// TIA Portal project "FactoryIO_Template" (V16)
// Vorlageprojekt für das Buch mit Zielsystem S7-1200

(* hardware
DEVICE "S7-1200-Station_1"  S7-1200 Station
   slot 0: "Baugruppenträger_0"  Rack  V1.0
   slot 1: "PLC_1"  CPU 1211C DC/DC/DC  6ES7 211-1AE40-0XB0  V4.1
*)

// ===== PLC "PLC_1"  CPU 1211C DC/DC/DC =====

VAR_GLOBAL   // PLC tag table "Standard-Variablentabelle"
   "Sensor_1" AT %I0.3 : Bool;
   "Sensor_2" AT %I0.4 : Bool;
   "Sensor_3" AT %I0.5 : Bool;
   "Start_Button" AT %I0.0 : Bool;
   "Stop_Button" AT %I0.1 : Bool;
   "Reset_Button" AT %I0.2 : Bool;
   "Sensor_Input" AT %I0.6 : Bool;
   "Sensor_Output" AT %I0.7 : Bool;
   "Limit_0" AT %I1.0 : Bool;
   "Limit_90" AT %I1.1 : Bool;
   "Conveyor_1_(C1)" AT %Q0.0 : Bool;
   "Conveyor_2_(C2)" AT %Q0.1 : Bool;
   "Conveyor_3_(C3)" AT %Q0.2 : Bool;
   "Conveyor_4_(C4)" AT %Q0.3 : Bool;
   "Roll_(+)" AT %Q0.4 : Bool;
   "Roll_(-)" AT %Q0.5 : Bool;
   "Turn" AT %Q0.6 : Bool;
   "Start_Light" AT %Q0.7 : Bool;
   "Stop_Light" AT %Q1.0 : Bool;
   "Long_Counter" AT %QD40 : DInt;
   "Medium_Counter" AT %QD44 : DInt;
   "Short_Counter" AT %QD48 : DInt;
   "Long" AT %M1.0 : Bool;
   "Medium" AT %M1.1 : Bool;
   "Short" AT %M1.2 : Bool;
   "Emitter" AT %Q1.1 : Bool;
   "Read_Long_Counter" AT %MD0 : DInt;
   "Read_Medium_Counter" AT %MD4 : DInt;
   "Read_Short_Counter" AT %MD8 : DInt;
END_VAR

DATA_BLOCK "Phan_Loai_DB"   // DB1
{ S7_Optimized_Access := 'TRUE' }
VERSION : 0.1
// stored: InstanceOfName Phan_Loai
"Phan_Loai"
BEGIN
END_DATA_BLOCK

DATA_BLOCK "Control_DB"   // DB2
{ S7_Optimized_Access := 'TRUE' }
VERSION : 0.1
// stored: InstanceOfName Control
"Control"
BEGIN
END_DATA_BLOCK

// folder: System blocks/Program resources

DATA_BLOCK "Delay_500ms"   // DB3
{ S7_Optimized_Access := 'TRUE' }
AUTHOR : Simatic
FAMILY : IEC
NAME : IEC_TMR
VERSION : 1.0
// stored: InstanceOfName IEC_TIMER
"IEC_TIMER"
BEGIN
END_DATA_BLOCK

DATA_BLOCK "Counter_Long"   // DB4
{ S7_Optimized_Access := 'TRUE' }
AUTHOR : Simatic
FAMILY : IEC
NAME : CNTR
VERSION : 1.0
// stored: InstanceOfName IEC_COUNTER
"IEC_COUNTER"
BEGIN
END_DATA_BLOCK

DATA_BLOCK "Counter_Medium"   // DB5
{ S7_Optimized_Access := 'TRUE' }
AUTHOR : Simatic
FAMILY : IEC
NAME : CNTR
VERSION : 1.0
// stored: InstanceOfName IEC_COUNTER
"IEC_COUNTER"
BEGIN
END_DATA_BLOCK

DATA_BLOCK "Counter_Short"   // DB6
{ S7_Optimized_Access := 'TRUE' }
AUTHOR : Simatic
FAMILY : IEC
NAME : CNTR
VERSION : 1.0
// stored: InstanceOfName IEC_COUNTER
"IEC_COUNTER"
BEGIN
END_DATA_BLOCK

// folder: (top level)

FUNCTION_BLOCK "Phan_Loai"   // FB1, LAD
{ S7_Optimized_Access := 'TRUE' }
VERSION : 0.1
   VAR_INPUT
      SS1 : Bool;
      SS2 : Bool;
      SS3 : Bool;
   END_VAR
   VAR_OUTPUT
      Long : Bool;
      Medium : Bool;
      Short : Bool;
   END_VAR
   VAR
      Temp_Long : Bool;
      Temp_Medium : Bool;
      Temp_Short : Bool;
      Reset : Bool;
      Temp_1 : Bool;
      "A" : Bool;
      "B" : Bool;
      C : Bool;
      D : Bool;
      "E" : Bool;
   END_VAR
   VAR_TEMP   // added for the SCL form of the ladder/FBD networks
      _w1 : Bool;
   END_VAR
BEGIN

REGION Network 1: Long
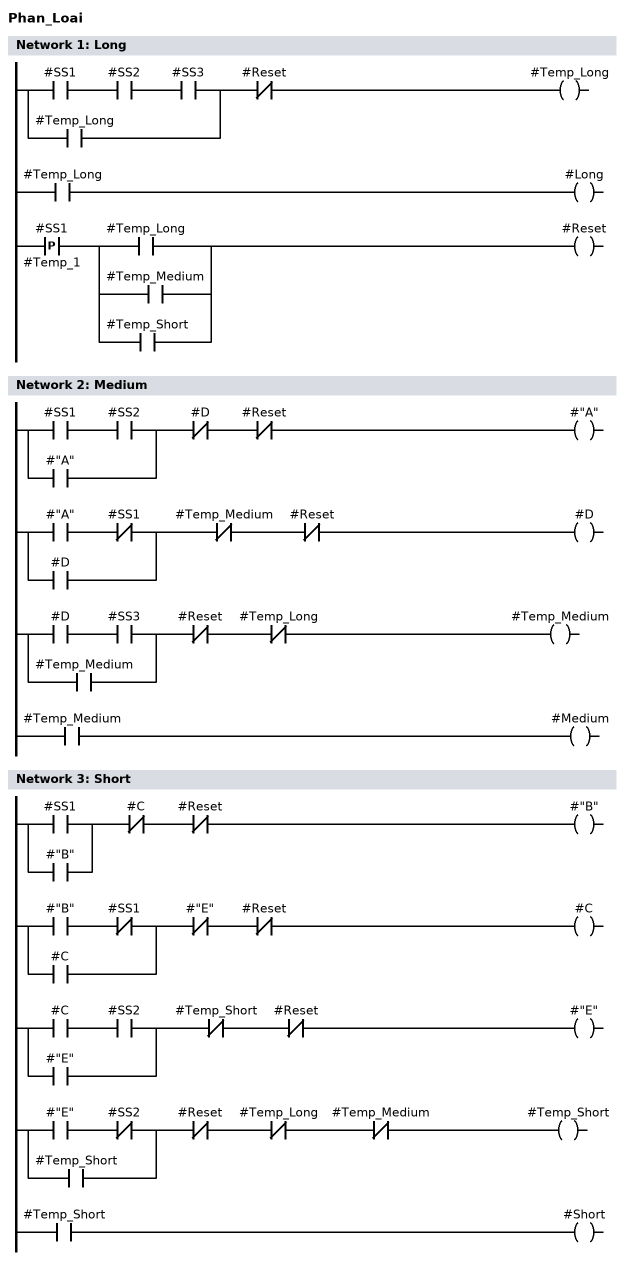
   RUNG wire#powerrail
      Contact( #SS1 )
      Contact( #SS2 )
      Contact( #SS3 )
      wire#w1
      I_Contact( #Reset )
      Coil( #Temp_Long )
   END_RUNG
   RUNG wire#powerrail
      Contact( #Temp_Long )
   END_RUNG wire#w1
   RUNG wire#powerrail
      Contact( #Temp_Long )
      Coil( #Long )
   END_RUNG
   RUNG wire#powerrail
      P_Contact(operand := #SS1, bit := #Temp_1)
      wire#w2
      Contact( #Temp_Long )
      wire#w3
      Coil( #Reset )
   END_RUNG
   RUNG wire#w2
      Contact( #Temp_Medium )
   END_RUNG wire#w3
   RUNG wire#w2
      Contact( #Temp_Short )
   END_RUNG wire#w3
   // the same network as SCL:
   #Temp_Long := ((#SS1 AND #SS2 AND #SS3) OR #Temp_Long) AND NOT #Reset;
   #Long := #Temp_Long;
   #_w1 := #SS1 AND NOT #Temp_1;   // rising edge of #SS1
   #Temp_1 := #SS1;
   #Reset := #_w1 AND (#Temp_Long OR #Temp_Medium OR #Temp_Short);
END_REGION

REGION Network 2: Medium
   RUNG wire#powerrail
      Contact( #SS1 )
      Contact( #SS2 )
      wire#w1
      I_Contact( #D )
      I_Contact( #Reset )
      Coil( #"A" )
   END_RUNG
   RUNG wire#powerrail
      Contact( #"A" )
   END_RUNG wire#w1
   RUNG wire#powerrail
      Contact( #"A" )
      I_Contact( #SS1 )
      wire#w2
      I_Contact( #Temp_Medium )
      I_Contact( #Reset )
      Coil( #D )
   END_RUNG
   RUNG wire#powerrail
      Contact( #D )
   END_RUNG wire#w2
   RUNG wire#powerrail
      Contact( #D )
      Contact( #SS3 )
      wire#w3
      I_Contact( #Reset )
      I_Contact( #Temp_Long )
      Coil( #Temp_Medium )
   END_RUNG
   RUNG wire#powerrail
      Contact( #Temp_Medium )
   END_RUNG wire#w3
   RUNG wire#powerrail
      Contact( #Temp_Medium )
      Coil( #Medium )
   END_RUNG
   // the same network as SCL:
   #"A" := ((#SS1 AND #SS2) OR #"A") AND NOT #D AND NOT #Reset;
   #D := ((#"A" AND NOT #SS1) OR #D) AND NOT #Temp_Medium AND NOT #Reset;
   #Temp_Medium := ((#D AND #SS3) OR #Temp_Medium) AND NOT #Reset AND NOT #Temp_Long;
   #Medium := #Temp_Medium;
END_REGION

REGION Network 3: Short
   RUNG wire#powerrail
      Contact( #SS1 )
      wire#w1
      I_Contact( #C )
      I_Contact( #Reset )
      Coil( #"B" )
   END_RUNG
   RUNG wire#powerrail
      Contact( #"B" )
   END_RUNG wire#w1
   RUNG wire#powerrail
      Contact( #"B" )
      I_Contact( #SS1 )
      wire#w2
      I_Contact( #"E" )
      I_Contact( #Reset )
      Coil( #C )
   END_RUNG
   RUNG wire#powerrail
      Contact( #C )
   END_RUNG wire#w2
   RUNG wire#powerrail
      Contact( #C )
      Contact( #SS2 )
      wire#w3
      I_Contact( #Temp_Short )
      I_Contact( #Reset )
      Coil( #"E" )
   END_RUNG
   RUNG wire#powerrail
      Contact( #"E" )
   END_RUNG wire#w3
   RUNG wire#powerrail
      Contact( #"E" )
      I_Contact( #SS2 )
      wire#w4
      I_Contact( #Reset )
      I_Contact( #Temp_Long )
      I_Contact( #Temp_Medium )
      Coil( #Temp_Short )
   END_RUNG
   RUNG wire#powerrail
      Contact( #Temp_Short )
   END_RUNG wire#w4
   RUNG wire#powerrail
      Contact( #Temp_Short )
      Coil( #Short )
   END_RUNG
   // the same network as SCL:
   #"B" := (#SS1 OR #"B") AND NOT #C AND NOT #Reset;
   #C := ((#"B" AND NOT #SS1) OR #C) AND NOT #"E" AND NOT #Reset;
   #"E" := ((#C AND #SS2) OR #"E") AND NOT #Temp_Short AND NOT #Reset;
   #Temp_Short := ((#"E" AND NOT #SS2) OR #Temp_Short) AND NOT #Reset AND NOT #Temp_Long AND NOT #Temp_Medium;
   #Short := #Temp_Short;
END_REGION
END_FUNCTION_BLOCK

FUNCTION_BLOCK "Control"   // FB2, LAD
{ S7_Optimized_Access := 'TRUE' }
VERSION : 0.1
   VAR_INPUT
      Long : Bool;
      Medium : Bool;
      Short : Bool;
      Start_Button : Bool;
      Stop_Button : Bool;
      Reset_Button : Bool;
      Sensor_Input : Bool;
      Sensor_Output : Bool;
      Limit_0 : Bool;
      Limit_90 : Bool;
   END_VAR
   VAR_OUTPUT
      "Conveyor_1_(C1)" : Bool;
      "Conveyor_2_(C2)" : Bool;
      "Conveyor_3_(C3)" : Bool;
      "Conveyor_4_(C4)" : Bool;
      "Roll_(+)" : Bool;
      "Roll_(-)" : Bool;
      Turn : Bool;
      Long_Counter : DInt;
      Medium_Counter : DInt;
      Short_Counter : DInt;
   END_VAR
   VAR
      C1_Temp : Bool;
      C_Temp : Bool;
      "A" : Bool;
      "Control_Roll_(+)" : Bool;
      "B" : Bool;
      C : Bool;
      Control_Turn : Bool;
      D : Bool;
      "E" : Bool;
      F : Bool;
      "Control_Roll_(-)" : Bool;
      G : Bool;
      H : Bool;
      I : Bool;
      K : Bool;
   END_VAR
   VAR_TEMP   // added for the SCL form of the ladder/FBD networks
      _w1 : Bool;
      _w2 : Bool;
      _w3 : Bool;
      _w4 : Bool;
      _w5 : Bool;
      _w6 : Bool;
      _w7 : Bool;
   END_VAR
BEGIN

REGION Network 1: Start up
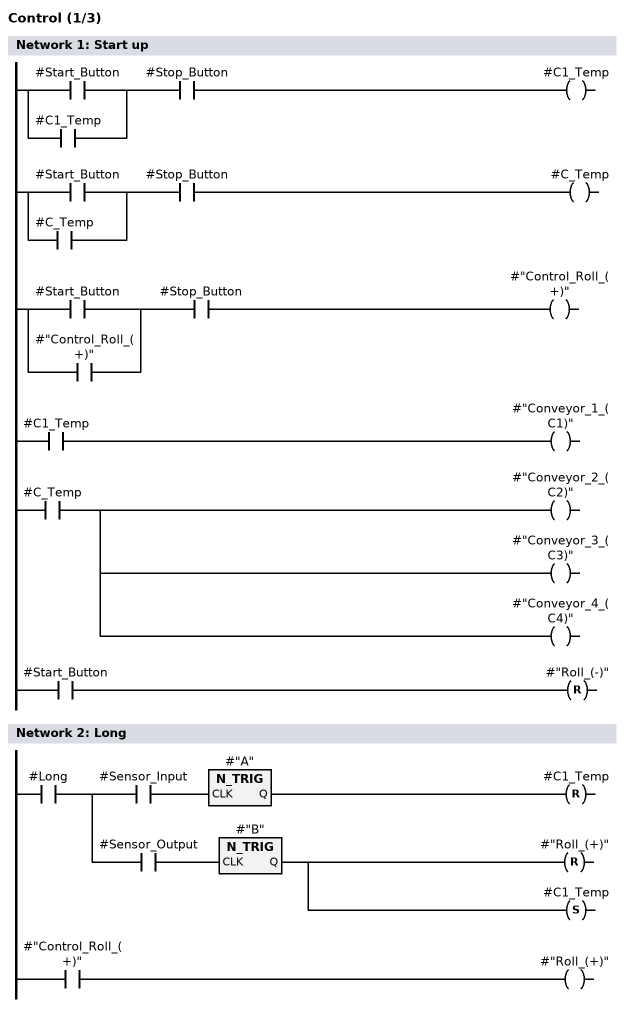
   RUNG wire#powerrail
      Contact( #Start_Button )
      wire#w1
      Contact( #Stop_Button )
      Coil( #C1_Temp )
   END_RUNG
   RUNG wire#powerrail
      Contact( #C1_Temp )
   END_RUNG wire#w1
   RUNG wire#powerrail
      Contact( #Start_Button )
      wire#w2
      Contact( #Stop_Button )
      Coil( #C_Temp )
   END_RUNG
   RUNG wire#powerrail
      Contact( #C_Temp )
   END_RUNG wire#w2
   RUNG wire#powerrail
      Contact( #Start_Button )
      wire#w3
      Contact( #Stop_Button )
      Coil( #"Control_Roll_(+)" )
   END_RUNG
   RUNG wire#powerrail
      Contact( #"Control_Roll_(+)" )
   END_RUNG wire#w3
   RUNG wire#powerrail
      Contact( #C1_Temp )
      Coil( #"Conveyor_1_(C1)" )
   END_RUNG
   RUNG wire#powerrail
      Contact( #C_Temp )
      wire#w4
      Coil( #"Conveyor_2_(C2)" )
   END_RUNG
   RUNG wire#w4
      Coil( #"Conveyor_3_(C3)" )
   END_RUNG
   RUNG wire#w4
      Coil( #"Conveyor_4_(C4)" )
   END_RUNG
   RUNG wire#powerrail
      Contact( #Start_Button )
      R_Coil( #"Roll_(-)" )
   END_RUNG
   // the same network as SCL:
   #C1_Temp := (#Start_Button OR #C1_Temp) AND #Stop_Button;
   #C_Temp := (#Start_Button OR #C_Temp) AND #Stop_Button;
   #"Control_Roll_(+)" := (#Start_Button OR #"Control_Roll_(+)") AND #Stop_Button;
   #"Conveyor_1_(C1)" := #C1_Temp;
   #"Conveyor_2_(C2)" := #C_Temp;
   #"Conveyor_3_(C3)" := #C_Temp;
   #"Conveyor_4_(C4)" := #C_Temp;
   IF #Start_Button THEN #"Roll_(-)" := FALSE; END_IF;
END_REGION

REGION Network 2: Long
   RUNG wire#powerrail
      Contact( #Long )
      wire#w1
      Contact( #Sensor_Input )
      N_Trig( #"A" )
      R_Coil( #C1_Temp )
   END_RUNG
   RUNG wire#w1
      Contact( #Sensor_Output )
      N_Trig( #"B" )
      wire#w2
      R_Coil( #"Roll_(+)" )
   END_RUNG
   RUNG wire#w2
      S_Coil( #C1_Temp )
   END_RUNG
   RUNG wire#powerrail
      Contact( #"Control_Roll_(+)" )
      Coil( #"Roll_(+)" )
   END_RUNG
   // the same network as SCL:
   #_w1 := #Long AND #Sensor_Input;
   #_w2 := NOT #_w1 AND #"A";   // falling edge
   #"A" := #_w1;
   IF #_w2 THEN #C1_Temp := FALSE; END_IF;
   #_w3 := #Long AND #Sensor_Output;
   #_w4 := NOT #_w3 AND #"B";   // falling edge
   #"B" := #_w3;
   IF #_w4 THEN
       #"Roll_(+)" := FALSE;
       #C1_Temp := TRUE;
   END_IF;
   #"Roll_(+)" := #"Control_Roll_(+)";
END_REGION

REGION Network 3: Medium
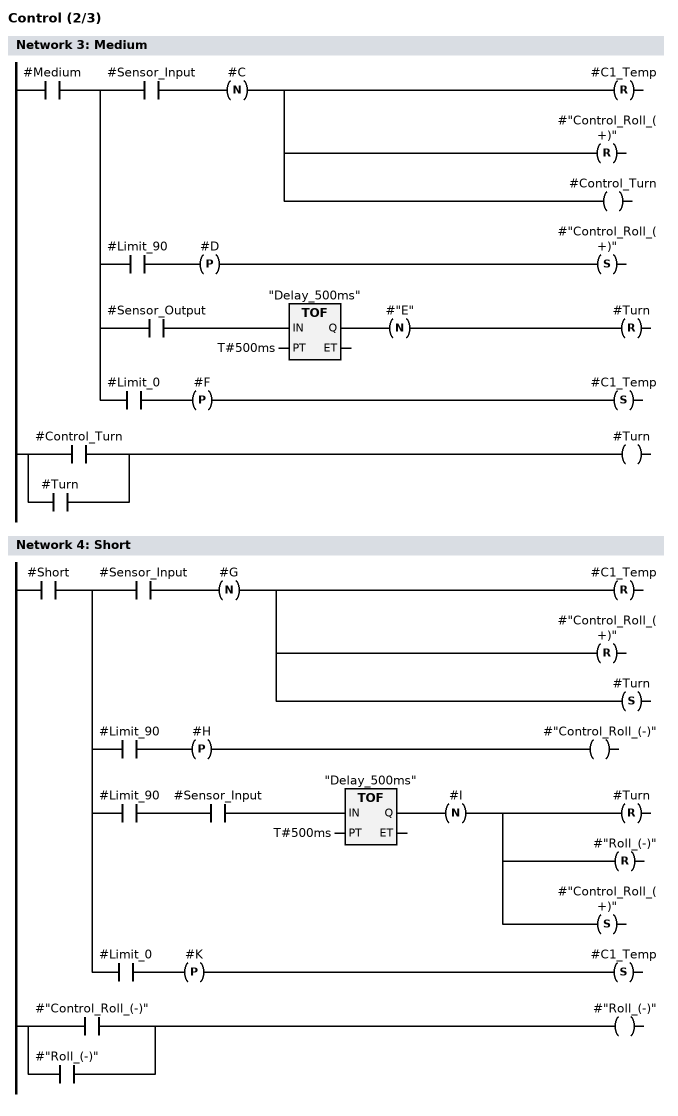
   #_w1 := #Medium AND #Sensor_Input;
   #_w2 := NOT #_w1 AND #C;   // falling edge
   #C := #_w1;
   IF #_w2 THEN
       #C1_Temp := FALSE;
       #"Control_Roll_(+)" := FALSE;
   END_IF;
   #Control_Turn := #_w2;
   #_w3 := #Medium AND #Limit_90;
   #_w4 := #_w3 AND NOT #D;   // rising edge
   #D := #_w3;
   IF #_w4 THEN #"Control_Roll_(+)" := TRUE; END_IF;
   "Delay_500ms".TOF(IN := #Medium AND #Sensor_Output, PT := T#500ms);
   #_w5 := NOT "Delay_500ms".Q AND #"E";   // falling edge
   #"E" := "Delay_500ms".Q;
   IF #_w5 THEN #Turn := FALSE; END_IF;
   #_w6 := #Medium AND #Limit_0;
   #_w7 := #_w6 AND NOT #F;   // rising edge
   #F := #_w6;
   IF #_w7 THEN #C1_Temp := TRUE; END_IF;
   #Turn := #Control_Turn OR #Turn;
END_REGION

REGION Network 4: Short
   #_w1 := #Short AND #Sensor_Input;
   #_w2 := NOT #_w1 AND #G;   // falling edge
   #G := #_w1;
   IF #_w2 THEN
       #C1_Temp := FALSE;
       #"Control_Roll_(+)" := FALSE;
       #Turn := TRUE;
   END_IF;
   #_w3 := #Short AND #Limit_90;
   #_w4 := #_w3 AND NOT #H;   // rising edge
   #H := #_w3;
   #"Control_Roll_(-)" := #_w4;
   "Delay_500ms".TOF(IN := #Short AND #Limit_90 AND #Sensor_Input, PT := T#500ms);
   #_w5 := NOT "Delay_500ms".Q AND #I;   // falling edge
   #I := "Delay_500ms".Q;
   IF #_w5 THEN
       #Turn := FALSE;
       #"Roll_(-)" := FALSE;
       #"Control_Roll_(+)" := TRUE;
   END_IF;
   #_w6 := #Short AND #Limit_0;
   #_w7 := #_w6 AND NOT #K;   // rising edge
   #K := #_w6;
   IF #_w7 THEN #C1_Temp := TRUE; END_IF;
   #"Roll_(-)" := #"Control_Roll_(-)" OR #"Roll_(-)";
END_REGION

REGION Network 5: Counter
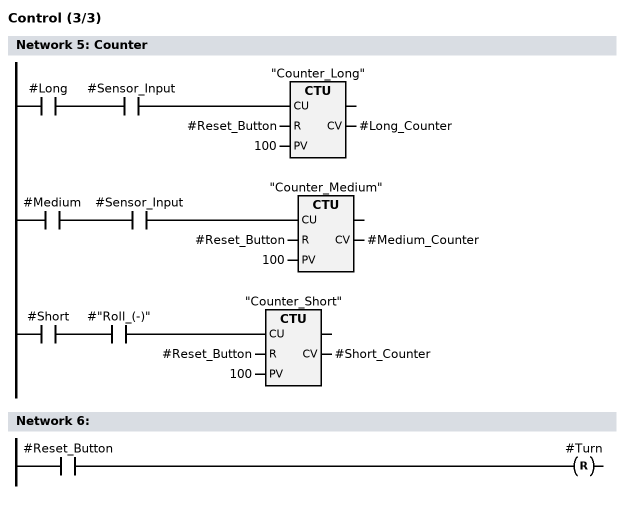
   "Counter_Long".CTU(CU := #Long AND #Sensor_Input, R := #Reset_Button, PV := 100, CV => #Long_Counter);
   "Counter_Medium".CTU(CU := #Medium AND #Sensor_Input, R := #Reset_Button, PV := 100, CV => #Medium_Counter);
   "Counter_Short".CTU(CU := #Short AND #"Roll_(-)", R := #Reset_Button, PV := 100, CV => #Short_Counter);
END_REGION

REGION Network 6
   RUNG wire#powerrail
      Contact( #Reset_Button )
      R_Coil( #Turn )
   END_RUNG
   // the same network as SCL:
   IF #Reset_Button THEN #Turn := FALSE; END_IF;
END_REGION
END_FUNCTION_BLOCK

FUNCTION "MHJ-PLC-Lab-Function-S71200" : Void   // FC9000, SCL
{ S7_Optimized_Access := 'TRUE' }
VERSION : 0.1
   VAR_TEMP
      rdTimeReturn : Int;
      outputTime : DTL;
      SyncVal : Byte;
      forVal : Int;
      forVal_2 : Int;
      Value : Byte;
   END_VAR
   VAR CONSTANT
      CompVal : Byte := 16#34;
      Value_01 : Byte := 16#11;
      Value_01_DW : DWord := 16#A165_D992;
      Value_02_DW : DWord := 16#58BE_4401;
   END_VAR
BEGIN

   #Value:=PEEK(area := 16#82,
        dbNumber := 0,
        byteOffset := 511);
   #Value := #Value + 1;

   POKE(area := 16#82,
        dbNumber := 0,
        byteOffset := 511,
        value := #Value);

   POKE(area:=16#81,
        dbNumber:=0,
        byteOffset:=1016,
        value:=#Value_01_DW);
   POKE(area := 16#81,
        dbNumber := 0,
        byteOffset := 1020,
        value := #Value_02_DW);

   POKE(area := 16#81,
        dbNumber := 0,
        byteOffset := 511,
        value := B#16#00);

   FOR #forVal := 0 TO 120 DO
       FOR #forVal_2:=0 TO 10 DO
           #rdTimeReturn:=RD_SYS_T(#outputTime);
           #rdTimeReturn := WR_SYS_T(#outputTime);
           #rdTimeReturn := RD_SYS_T(#outputTime);
           #rdTimeReturn := WR_SYS_T(#outputTime);
       END_FOR;
       #SyncVal:= PEEK(area := 16#81,
                      dbNumber := 0,
                      byteOffset := 511);
       IF #SyncVal = #CompVal THEN
          GOTO M_1;
       END_IF;
   END_FOR;
   RETURN;

   M_1:
   POKE(area := 16#81,
        dbNumber := 0,
        byteOffset := 511,
        value := B#16#0);
END_FUNCTION

ORGANIZATION_BLOCK "Main"   // OB1, FBD, ProgramCycle
TITLE = "Main Program Sweep (Cycle)"
{ S7_Optimized_Access := 'TRUE' }
VERSION : 0.1
   VAR_INPUT
      Initial_Call : Bool;   // Initial call of this OB
      Remanence : Bool;   // =True, if remanent data are available
   END_VAR
BEGIN

REGION Network 1: Konnektierungsbaustein für PLC-Lab
   // Im Netzwerk 1 wird der Konnektierungsbaustein für PLC-Lab aufgerufen.
   // Dieser Aufruf darf nicht entfernt werden!
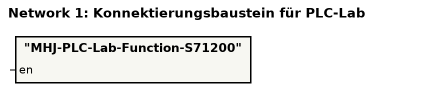
   "MHJ-PLC-Lab-Function-S71200"();
END_REGION

REGION Network 2: Ihr Programm
   // Schreiben Sie ab Netzwerk 2 Ihr Programm
END_REGION
END_ORGANIZATION_BLOCK

ORGANIZATION_BLOCK "control_system"   // OB123, LAD, ProgramCycle
TITLE = "Main Program Sweep (Cycle)"
{ S7_Optimized_Access := 'TRUE' }
VERSION : 0.1
   VAR_INPUT
      Initial_Call : Bool;   // Initial call of this OB
      Remanence : Bool;   // =True, if remanent data are available
   END_VAR
BEGIN

REGION Network 1: Phan loai san Pham
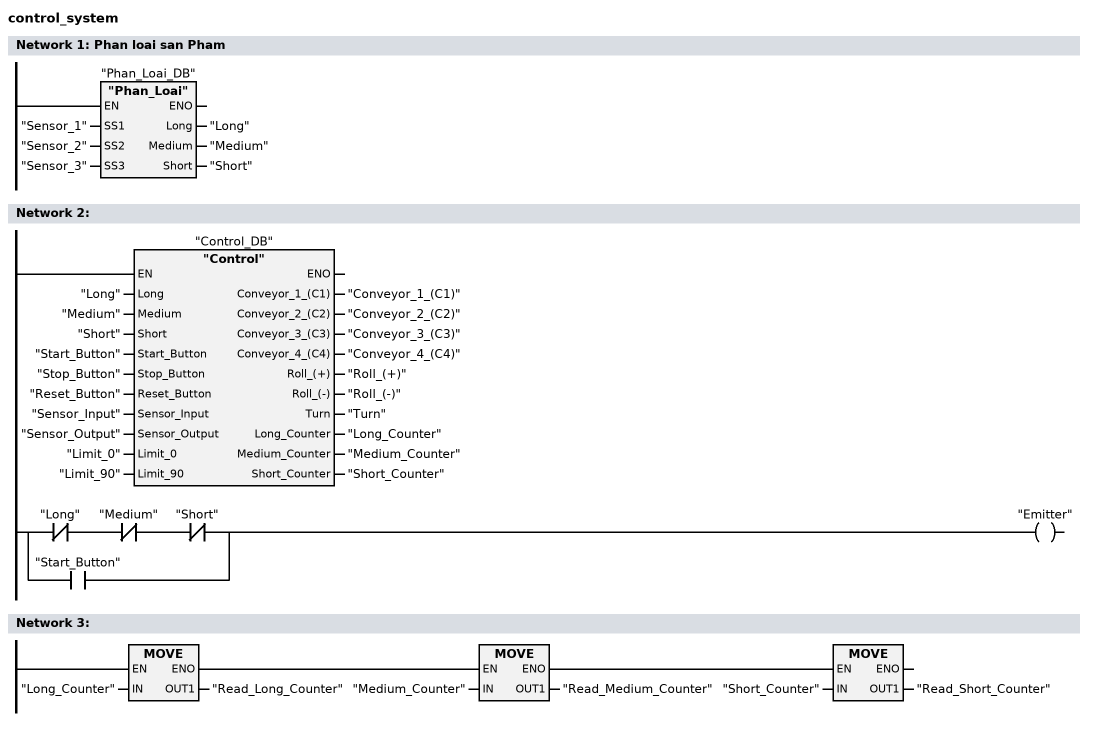
   RUNG wire#powerrail
      "Phan_Loai_DB"(SS1 := "Sensor_1", SS2 := "Sensor_2", SS3 := "Sensor_3", Long => "Long", Medium => "Medium", Short => "Short")
   END_RUNG
   // the same network as SCL:
   "Phan_Loai_DB"(SS1 := "Sensor_1",   // "Phan_Loai"
                  SS2 := "Sensor_2",
                  SS3 := "Sensor_3",
                  Long => "Long",
                  Medium => "Medium",
                  Short => "Short");
END_REGION

REGION Network 2
   RUNG wire#powerrail
      "Control_DB"(Long := "Long", Medium := "Medium", Short := "Short", Start_Button := "Start_Button", Stop_Button := "Stop_Button", Reset_Button := "Reset_Button", Sensor_Input := "Sensor_Input", Sensor_Output := "Sensor_Output", Limit_0 := "Limit_0", Limit_90 := "Limit_90", "Conveyor_1_(C1)" => "Conveyor_1_(C1)", "Conveyor_2_(C2)" => "Conveyor_2_(C2)", "Conveyor_3_(C3)" => "Conveyor_3_(C3)", "Conveyor_4_(C4)" => "Conveyor_4_(C4)", "Roll_(+)" => "Roll_(+)", "Roll_(-)" => "Roll_(-)", Turn => "Turn", Long_Counter => "Long_Counter", Medium_Counter => "Medium_Counter", Short_Counter => "Short_Counter")
   END_RUNG
   RUNG wire#powerrail
      I_Contact( "Long" )
      I_Contact( "Medium" )
      I_Contact( "Short" )
      wire#w1
      Coil( "Emitter" )
   END_RUNG
   RUNG wire#powerrail
      Contact( "Start_Button" )
   END_RUNG wire#w1
   // the same network as SCL:
   "Control_DB"(Long := "Long",   // "Control"
                Medium := "Medium",
                Short := "Short",
                Start_Button := "Start_Button",
                Stop_Button := "Stop_Button",
                Reset_Button := "Reset_Button",
                Sensor_Input := "Sensor_Input",
                Sensor_Output := "Sensor_Output",
                Limit_0 := "Limit_0",
                Limit_90 := "Limit_90",
                "Conveyor_1_(C1)" => "Conveyor_1_(C1)",
                "Conveyor_2_(C2)" => "Conveyor_2_(C2)",
                "Conveyor_3_(C3)" => "Conveyor_3_(C3)",
                "Conveyor_4_(C4)" => "Conveyor_4_(C4)",
                "Roll_(+)" => "Roll_(+)",
                "Roll_(-)" => "Roll_(-)",
                Turn => "Turn",
                Long_Counter => "Long_Counter",
                Medium_Counter => "Medium_Counter",
                Short_Counter => "Short_Counter");
   "Emitter" := (NOT "Long" AND NOT "Medium" AND NOT "Short") OR "Start_Button";
END_REGION

REGION Network 3
   RUNG wire#powerrail
      Move(in := "Long_Counter", out1 => "Read_Long_Counter")
      Move(in := "Medium_Counter", out1 => "Read_Medium_Counter")
      Move(in := "Short_Counter", out1 => "Read_Short_Counter")
   END_RUNG
   // the same network as SCL:
   "Read_Long_Counter" := "Long_Counter";
   "Read_Medium_Counter" := "Medium_Counter";
   "Read_Short_Counter" := "Short_Counter";
END_REGION
END_ORGANIZATION_BLOCK